FUNCTION_BLOCK FB_Queue
VAR_INPUT
END_VAR
VAR_OUTPUT
	bFull	 				:BOOL := FALSE;					// True if queue is full
	iNoOfEntries			:UINT := 0;						// Number of entries in the queue
	iNoOfFree				:UINT := cQueueSize; // Number of free entries
END_VAR
VAR
	iInputIndex 			:UINT := 1;						// Points to next input entry in queue
	iOutputIndex	 		:UINT := 1;						// Points to next output entry in queue
 	arrQueue	 			:ARRAY[1..cQueueSize] OF INT;	// Queue
	bError					:BOOL;							// True if error occurs
END_VAR
VAR CONSTANT
	cQueueSize				:UINT := 100;				
END_VAR

METHOD M_Flush : BOOL
VAR_INPUT
END_VAR
VAR
	iEntryEmpty		:INT;			// Entry with zero content
	iForIndex		:INT;			// Index used in for-loops	
END_VAR

// Flush Queue. All entries are deleted. Index's and counters are reset.
//----------------------------------------------------------------------

// Initialize empty entry
iEntryEmpty := 0;

// Reset all entries in queue
FOR iForIndex := 1 TO UINT_TO_INT(cQueueSize) BY 1 DO
	arrQueue[iForIndex] := iEntryEmpty;
END_FOR

// Reset index's and counters
iInputIndex 	:= 1;
iOutputIndex	:= 1;
iNoOfEntries	:= 0;
iNoOfFree		:= cQueueSize;
END_METHOD

METHOD M_GetEntry : BOOL
VAR_OUTPUT
	iEntry 				:INT;			// Value for found entry in queue 
	bNewEntry			:BOOL;			// True if new entry was foud in queue, False if queue is empty
END_VAR

// Check if there are any events in queue
IF(iInputIndex <> iOutputIndex ) THEN							
	// Min one event in queue, get next event
	iEntry := arrQueue[iOutputIndex];		
	bNewEntry := TRUE;
											
	// Update output index	
  	IF(iOutputIndex > (cQueueSize-1)) THEN 									
  		iOutputIndex := 1;
  	ELSE
		iOutputIndex := iOutputIndex + 1;
	END_IF
	
	// Update the entry counter
	iNoOfEntries := iNoOfEntries - 1;
	
	// Reset full flag if it was set
	bFull := FALSE; 
ELSE
	// No events in queue
	bNewEntry := FALSE;
	iNoOfEntries := 0;
END_IF;

// Update count for number of free entires
iNoOfFree := cQueueSize - iNoOfEntries;
END_METHOD

METHOD M_GetFullStatus : BOOL
VAR_INPUT
END_VAR
// Returns true if queue is full

// Initialize to false
M_GetFullStatus := FALSE;

// Update signal
IF((iInputIndex+1) > cQueueSize) THEN
	// Input index will loop around at next entry. Make sure that output index is not occuping this place.
	IF iOutputIndex = 0 THEN
		M_GetFullStatus := TRUE;
	END_IF
ELSIF ((iInputIndex + 1) = iOutputIndex) THEN
	// Output is occuping next entry. Queue full 
	M_GetFullStatus := TRUE;
END_IF

// Check entry counter	
IF iNoOfEntries >= cQueueSize THEN
	M_GetFullStatus := TRUE;
END_IF
END_METHOD

METHOD M_PutEntry : BOOL
VAR_INPUT
	iEntry	 		:INT;			// Value to be stored in queue
END_VAR

// Update Full flag
IF iNoOfEntries >= cQueueSize THEN
	bFull := TRUE;
ELSE
	bFull := FALSE;
END_IF


// Put entry into queue unless it is full
IF NOT bFull THEN
	arrQueue[iInputIndex] := iEntry;
	iNoOfEntries := iNoOfEntries + 1;
	IF iNoOfEntries > cQueueSize THEN
		bError := TRUE;
	END_IF 
END_IF

// Update input index and find out if queue is full
// bFull := FALSE;
IF((iInputIndex+1) > cQueueSize) THEN
	// Input index has reached end of queue => loop back
	IF(iOutputIndex <> 1 )  THEN
		// Output index is NOT occuping the first index
   		iInputIndex := 1;
  	ELSE
    	// Output index IS occuping the first index => Queue full
		bFull := TRUE;
	 END_IF
ELSE
	// Input index has NOT reach end of queue
	IF((iInputIndex + 1) <> iOutputIndex) THEN
		iInputIndex := iInputIndex + 1;
  	ELSE
		bFull := TRUE;
	END_IF
END_IF

// Update count for number of free entires
iNoOfFree := cQueueSize - iNoOfEntries;
END_METHOD

END_FUNCTION_BLOCK

(* stored: Version 1.1.0.1, ProductVersion 3.1.4024.12
   POU FB_Queue: Id {c5f56251-4456-43d5-80bc-17cb2949ea14}, SpecialFunc None
   Method M_Flush: Id {ad25ed7e-5d54-42d6-af0d-2a50f2a396bf}
   Method M_GetEntry: Id {d55c21b4-2b5e-44b2-885f-261fd9358c6f}
   Method M_GetFullStatus: Id {40ad2313-58bd-4dce-8544-9770ed6a1c62}
   Method M_PutEntry: Id {e8c7d225-3dfb-4b80-a9e1-4e9eb329f4fd} *)
